FUNCTION_BLOCK RunAxis
VAR_INPUT
END_VAR
VAR_OUTPUT
	PositionFeedback : LREAL;
END_VAR
VAR_IN_OUT
	Comm : AxisBase; // public interface
END_VAR
VAR	
	Axis : AXIS_REF;
	 
	fbMoveAbs : MC_MoveAbsolute;
	fbMoveHome : MC_Home;
	fbPower : MC_Power;
	fbReset: MC_Reset;
	
	//Status reading
	fbReadParameter: MC_ReadParameter;
	fbReadActualPosition : MC_ReadActualPosition;
	fbReadStatus : MC_ReadStatus;
END_VAR

fbMoveAbs(
	Axis:= Axis, 
	Execute:= , 
	Position:= , 
	Velocity:= , 
	Acceleration:= , 
	Deceleration:= , 
	Jerk:= , 
	BufferMode:= , 
	Options:= , 
	Done=> , 
	Busy=> , 
	Active=> , 
	CommandAborted=> , 
	Error=> , 
	ErrorID=> );
	
fbMoveHome(
	Axis:= Axis, 
	Execute:= , 
	Position:= , 
	HomingMode:= , 
	BufferMode:= , 
	Options:= , 
	bCalibrationCam:= , 
	Done=> , 
	Busy=> , 
	Active=> , 
	CommandAborted=> , 
	Error=> , 
	ErrorID=> );
	
fbPower(
	Axis:= Axis, 
	Enable:= , 
	Enable_Positive:= , 
	Enable_Negative:= , 
	Override:= , 
	BufferMode:= , 
	Options:= , 
	Status=> , 
	Busy=> , 
	Active=> , 
	Error=> , 
	ErrorID=> );
	
fbReset(
	Axis:= Axis, 
	Execute:= , 
	Done=> , 
	Busy=> , 
	Error=> , 
	ErrorID=> );
	
//Status reading and update
fbReadParameter(
	Axis:= Axis, 
	Enable:= TRUE, 
	ParameterNumber:= ActualVelocity, 
	ReadMode:= , 
	Valid=> , 
	Busy=> , 
	Error=> , 
	ErrorID=> , 
	Value=> );
comm.SPD_FEEDBACK := LREAL_TO_DWORD(fbReadParameter.Value*1000);
fbReadParameter(
	Axis:= Axis, 
	Enable:= TRUE, 
	ParameterNumber:= CommandedPosition, 
	ReadMode:= , 
	Valid=> , 
	Busy=> , 
	Error=> , 
	ErrorID=> , 
	Value=> );
comm.POS_COMMAND := LREAL_TO_DWORD(fbReadParameter.Value*1000);
fbReadActualPosition(
	Axis:= axis, 
	Enable:= TRUE, 
	Valid=> , 
	Busy=> , 
	Error=> , 
	ErrorID=> , 
	Position=> PositionFeedback);
comm.POS_FEEDBACK := LREAL_TO_DWORD(PositionFeedback*1000);

fbReadStatus(
	Axis:= axis, 
	Enable:= TRUE, 
	Valid=> , 
	Busy=> , 
	Error=> , 
	ErrorID=> , 
	ErrorStop=> , 
	Disabled=> , 
	Stopping=> , 
	StandStill=> , 
	DiscreteMotion=> , 
	ContinuousMotion=> , 
	SynchronizedMotion=> , 
	Homing=> , 
	ConstantVelocity=> , 
	Accelerating=> , 
	Decelerating=> , 
	Status=> );

comm.MON_CONTROL_WORD.0 := fbPower.Enable; //servo on
comm.MON_CONTROL_WORD.15 := fbReset.Execute; // alarm clear
comm.RUN_STATUS.1 := fbReadStatus.StandStill; //run with servo on
comm.RUN_STATUS.3 := not fbReadStatus.Error; //Servo ready

METHOD ExecuteCommandBlock : BOOL
VAR_INPUT
	ptBlock : POINTER TO CommandBlockGeneric;
	execute : BOOL; //used to do mutex
END_VAR
VAR
	// Common Parameters
	speedInmm : LREAL;
	accInmms:LREAL;
	decInmms:LREAL;
	torqueLimitInPercentage:LREAL;
	//MC block routing
	ptMcExecute : POINTER TO BOOL;
	ptMcDone : POINTER TO BOOL;
	ptMcBusy : POINTER TO BOOL;
	ptMcError : POINTER TO BOOL;
END_VAR
VAR_OUTPUT
	done:bool;
END_VAR
//1. Do parameter translating
//2. Do command routing
//3. Control execute flow

IF NOT execute THEN
	RETURN;
END_IF

//parameter writing
speedInmm:=(LWORD_TO_LREAL(ptBlock^.base.SPEED)/1000);
accInmms:=((speedInmm)/(LWORD_TO_LREAL(ptBlock^.base.ACC_TIME)/1000));
decInmms:=((speedInmm)/(LWORD_TO_LREAL(ptBlock^.base.DEC_TIME)/1000));
torqueLimitInPercentage:=((LWORD_TO_LREAL(ptBlock^.base.TORQUE_LIMIT)/100));

//command routing
CASE ptBlock^.base.COMMAND_TYPE OF
eCommandTypes.POSITION:	
//Position command
ptMcExecute:=ADR(fbMoveAbs.Execute);
ptMcDone:=ADR(fbMoveAbs.Done);
ptMcBusy:=ADR(fbMoveAbs.Busy);
ptMcError:=ADR(fbMoveAbs.Error);

fbMoveAbs.Velocity := speedInmm;
//...
fbMoveAbs.Position := LWORD_TO_LREAL(ptBlock^.position.COORDINATE/1000); //

;
eCommandTypes.ZRET:
//Home command
ptMcExecute:=ADR(fbMoveHome.Execute);
ptMcDone:=ADR(fbMoveHome.Done);
ptMcBusy:=ADR(fbMoveHome.Busy);
ptMcError:=ADR(fbMoveHome.Error);
;
ELSE
	return;
END_CASE

//auto stop execute when error , would do raising edge again when error eliminated
ptMcExecute^ := NOT (ptMcError^) AND NOT (ptMcDone^);

done := ptMcDone^;

ExecuteCommandBlock:=done;
END_METHOD

METHOD FB_init : BOOL
VAR_INPUT
	bInitRetains : BOOL; // if TRUE, the retain variables are initialized (warm start / cold start)
	bInCopyCode : BOOL;  // if TRUE, the instance afterwards gets moved into the copy code (online change)
END_VAR
END_METHOD

END_FUNCTION_BLOCK

(* stored: Version 1.1.0.1, ProductVersion 3.1.4020.12
   POU RunAxis: Id {1e355049-017f-4f7f-88a6-a7040666a5c5}, SpecialFunc None
   Method ExecuteCommandBlock: Id {248fd65c-916e-4c41-b72b-91932f742cc7}
   Method FB_init: Id {5aeba573-47c3-411b-9f3d-8af6b6892223} *)
